// TIA Portal V18 export
// export: Created 2026-06-21T12:15:02Z, ExportSetting WithDefaults
PlcWatchTable "WT_PLC1_Main_Sequence"
  PlcWatchTableEntry "HMI_Sim_Mode"
  PlcWatchTableEntry "HMI_Run_Enable"
  PlcWatchTableEntry "HMI_Use_Sim_Input_PLC1"
  PlcWatchTableEntry "HMI_Use_Sim_Input_BonChua"
  PlcWatchTableEntry "Gia_Lap_Mat_Ket_Noi_HMI"
  PlcWatchTableEntry "HMI_Load_Default_Recipe"
  PlcWatchTableEntry "Nut_Khoi_Dong_HMI"
  PlcWatchTableEntry "Nut_Dung_HMI"
  PlcWatchTableEntry "Nut_Reset_HMI"
  PlcWatchTableEntry "Nut_EStop_HMI"
  PlcWatchTableEntry "PLC1_State"
  PlcWatchTableEntry "BonChua_State"
  PlcWatchTableEntry "PLC1_Loi_Tong"
  PlcWatchTableEntry "FQ3200_Bon1_HMI"
  PlcWatchTableEntry "LT3203_Bon1_HMI"
  PlcWatchTableEntry "FQ3205_Bon2_HMI"
  PlcWatchTableEntry "LT3209_Bon2_HMI"
  PlcWatchTableEntry "TT3208_Bon2_HMI"
  PlcWatchTableEntry "LT3302_BonChua1_HMI"
  PlcWatchTableEntry "TT3301_BonChua1_HMI"
  PlcWatchTableEntry "LT3307_BonChua2_HMI"
  PlcWatchTableEntry "PI3308_Truoc_Filter_HMI"
  PlcWatchTableEntry "FT3309_Xa_Thanh_Pham_HMI"
  PlcWatchTableEntry "V3230_Nuoc_Bon1"
  PlcWatchTableEntry "AGTR3260_Khuay_Bon1"
  PlcWatchTableEntry "V3235_Nuoc_Bon2"
  PlcWatchTableEntry "CV3206_Hoi_Bon2"
  PlcWatchTableEntry "VFD_Bon2_Run"
  PlcWatchTableEntry "VFD_Bon2_Dao_Chieu"
  PlcWatchTableEntry "Pump3264_Chuyen_Nhanh1"
  PlcWatchTableEntry "Pump3364_Filter"
  PlcWatchTableEntry "CV_Filler_Cap_Dich"
  PlcWatchTableEntry "HMI_Anim_Bon1_Frame"
  PlcWatchTableEntry "HMI_Anim_Bon2_Frame"
